INTERFACE I_ActivePower	// don't not EXTENDS I_ActivePowerNoFB, it violates Liskov Substitution Principle (LSP)

PROPERTY Active : reference to bool
GET
END_GET
END_PROPERTY

PROPERTY Busy : REFERENCE TO bool
GET
END_GET
END_PROPERTY

PROPERTY Error : reference to bool
GET
END_GET
END_PROPERTY

METHOD MR_Abort : bool
VAR_INPUT
END_VAR
END_METHOD

METHOD MR_Init : bool
VAR_INPUT
END_VAR
END_METHOD

METHOD MR_PowerOFF : BOOL
VAR_INPUT
END_VAR
END_METHOD

METHOD MR_PowerON : BOOL
VAR_INPUT
END_VAR
END_METHOD

METHOD MR_Reset : bool
VAR_INPUT
END_VAR
END_METHOD

(*Powerer on success*)
PROPERTY Powered : REFERENCE TO BOOL
GET
END_GET
END_PROPERTY

PROPERTY PowerOffIsCalled : bool
GET
END_GET
END_PROPERTY

PROPERTY PowerOnIsCalled : bool
GET
END_GET
END_PROPERTY

(*return value depedning on Request*)
PROPERTY ReasonError : string
GET
END_GET
END_PROPERTY

END_INTERFACE

(* stored: Version 1.1.0.1, ProductVersion 3.1.4024.12
   Itf I_ActivePower: Id {e4d392f5-3228-42b6-907b-ce95dee03de3}
   Property Active: Id {55fbb479-5223-4482-b7af-3105728ac033}
   Get Get: Id {3d521bad-d28b-4fd1-8e3f-a03de628cad5}
   Property Busy: Id {eacde2af-5819-4e39-ac27-2a6ec58a903b}
   Get Get: Id {dcaa9236-b632-4433-948b-c305fb30f045}
   Property Error: Id {646b5fa8-b6ab-4758-81c9-e18d4fb55467}
   Get Get: Id {735eb9f8-4253-4dcc-ab4a-989b9a1bce38}
   Method MR_Abort: Id {ed366470-69bd-4395-8c06-7ee3a8ea6308}
   Method MR_Init: Id {f3f2dbe3-7e7e-4064-8230-206aedab54a6}
   Method MR_PowerOFF: Id {fb6d8ace-5aaf-423b-ac19-721c502e3826}
   Method MR_PowerON: Id {2dbf883b-7cf2-4d79-816c-8ee157c39308}
   Method MR_Reset: Id {724598b8-ed33-4ba4-bb07-89d9ef6a61ec}
   Property Powered: Id {0ab80262-39ba-4135-9eec-c3b702ce9e37}
   Get Get: Id {cd02c1eb-0d30-4592-bb7a-a3607ce276d6}
   Property PowerOffIsCalled: Id {3de0dd29-91a2-46c6-abf3-5e4c21c2da7f}
   Get Get: Id {d6837f00-9360-4876-9c5e-b134773d5b71}
   Property PowerOnIsCalled: Id {e6e52be3-d24c-4b84-9646-aa73761429a4}
   Get Get: Id {353a6334-06a6-412a-9b39-37a7f939d411}
   Property ReasonError: Id {54e89aaa-963a-4230-b420-ea58a55c43af}
   Get Get: Id {22ea26c3-cc11-40f1-9ae7-6f7efa0688ea} *)
